// TIA Portal V20 export
// export: Created 2026-07-10T11:12:35.0422009Z, ExportSetting WithDefaults, DisplayName Totally Integrated Automation Portal, DisplayVersion V20, DisplayName TIA Portal Openness, DisplayVersion V20, DisplayName TIA Portal Version Control Interface, DisplayVersion V20, DisplayName STEP 7 Professional, DisplayVersion V20, DisplayName STEP 7 Safety, DisplayVersion V20, DisplayName WinCC Basic/Comfort/Advanced, DisplayVersion V20, DisplayName WinCC Unified, DisplayVersion V20
FUNCTION_BLOCK "ChlorationCalculate"   // FB7, SCL
{ S7_Optimized_Access := 'TRUE' }
VERSION : 0.1
// stored: AutoNumber true, IsIECCheckEnabled false, IsRetainMemResEnabled false, MemoryReserve 100, SetENOAutomatically false, UDAEnableTagReadback false
   VAR_INPUT
      measuredChlorine : Real;
   END_VAR
   VAR_IN_OUT
      ChlorationParams : Struct
         SetpointMin : Real;
         SetpointMax : Real;
         BaseDose : Real;
         ActualDose : Real;
         DoseChangeMax : Real;
         DosingMin : Real;
         DosingMax : Real;
         CorectionCoef : Real;
      END_STRUCT;
   END_VAR
   VAR RETAIN
      setpointDeviation : Real;
      doseCorection : Real := 1.0;
      doseCorectionOld : Real := 1.0;
   END_VAR
   VAR
      doseChangeMaxReal : Real;
   END_VAR
BEGIN
   IF NOT "MB".Table.ChangeChlorMeasure THEN
       RETURN;
   END_IF;

   IF #measuredChlorine <= "MB".Table.Chlor_SetpointMin OR
       #measuredChlorine >= "MB".Table.Chlor_SetpointMax THEN

       #setpointDeviation := ((("MB".Table.Chlor_SetpointMax + "MB".Table.Chlor_SetpointMin) / 2) - #measuredChlorine)* "MB".Table.Chlor_Corection;

       #doseCorection := #doseCorectionOld * (1 + #setpointDeviation);

       #doseChangeMaxReal := #ChlorationParams.DoseChangeMax / 100;

       IF #doseCorection - #doseCorectionOld > #doseChangeMaxReal THEN
           #doseCorection := #doseCorectionOld * (1 + #doseChangeMaxReal);
       ELSIF #doseCorection - #doseCorectionOld < - (#doseChangeMaxReal) THEN
           #doseCorection := #doseCorectionOld * (1 - #doseChangeMaxReal);
       END_IF;

       #ChlorationParams.ActualDose := "MB".Table.Chlor_BaseDose * #doseCorection;

       IF #ChlorationParams.ActualDose >= #ChlorationParams.DosingMax THEN
           #doseCorection := #ChlorationParams.DosingMax / "MB".Table.Chlor_BaseDose;
           #ChlorationParams.ActualDose := "MB".Table.Chlor_BaseDose * #doseCorection;
       ELSIF #ChlorationParams.ActualDose <= #ChlorationParams.DosingMin THEN
           #doseCorection := #ChlorationParams.DosingMin / "MB".Table.Chlor_BaseDose;
           #ChlorationParams.ActualDose := "MB".Table.Chlor_BaseDose * #doseCorection;
       END_IF;

       #doseCorectionOld := #doseCorection;

   END_IF;
END_FUNCTION_BLOCK
